{attribute 'OPC.UA.DA' := '0'}
TYPE ResponsivityConfig :
STRUCT
	Responsivity_mA_W : LREAL;
END_STRUCT
END_TYPE

(* stored: Version 1.1.0.1, ProductVersion 3.1.4024.10
   DUT ResponsivityConfig: Id {de4da026-0d11-4569-8c88-ca93d4d1ea22} *)
